Fanuc KAREL source: CURPOS.kl

PROGRAM T
%NOLOCKGROUP
VAR
 v0 : INTEGER
 v1 : INTEGER
 v2 : INTEGER
 res : XYZWPREXT
BEGIN
 res = CURPOS(v0, v1, v2)
END T
